// TwinCAT 3 PLC project ArbiterPLC
// ProgramVersion: 3.1.4022.7
// libraries:
//   Tc2_MC2, * (Beckhoff Automation GmbH)
//   Tc2_Standard, * (Beckhoff Automation GmbH)
//   Tc2_System, * (Beckhoff Automation GmbH)
//   Tc2_SystemCX, * (Beckhoff Automation GmbH)
//   Tc2_Utilities, * (Beckhoff Automation GmbH)
//   Tc3_Module, * (Beckhoff Automation GmbH)
//   LCLS General,newest,SLAC
//   PMPS,0.0.0,SLAC - LCLS
// project tree:
//   / FFOTask.TcTTO, PlcTask.TcTTO
//   GVLs/ GVL.TcGVL, GVL_CheckBounds.TcGVL
//   ImplicitChecks/ CheckBounds.TcPOU, CheckRangeSigned.TcPOU, CheckRangeUnsigned.TcPOU
//   POUs/Accelerator/ FB_Hgvpu.TcPOU, FB_SXU.TcPOU, FB_UndulatorSegment.TcPOU
//   POUs/ CurrentBPUpdate.TcPOU, CXDisplay.TcPOU, Fast_Faults_Evaluate.TcPOU, FB_BPControlDevice.TcPOU, FB_eVSimulator.TcPOU, FB_StopperWatcher.TcPOU, MachineSimulation.TcPOU, MAIN.TcPOU, PMPS_Arbiter.TcPOU, Testing.TcPOU
// real-time tasks:
//   TASK PlcTask: cycle T#10ms, priority 2, ADS port 350
//   TASK FFOTask: cycle T#1ms, priority 1, ADS port 351
// I/O:
//   DEVICE Device 1 (EtherCAT), AmsNetId 0.0.0.0.2.1
//     Term 12 (EK1200) [EK1200-5000 EtherCAT Power supply (2A E-Bus)]
//       FFO [EL2202 2Ch. Dig. Output 24V, 0.5A]
//       PMPS_Premp [EL2809 16Ch. Dig. Output 24V, 0.5A]
//       Term 12 (EK1122) [EK1122 2 port EtherCAT junction]
//         Term 13 (EK1100) [EK1100 EtherCAT Coupler (2A E-Bus)]
//           PPS_Stoppers [EL1008 8Ch. Dig. Input 24V, 3ms]
//           Term 15 (EL1008) [EL1008 8Ch. Dig. Input 24V, 3ms]
//           MPS_Relay [EL2004 4Ch. Dig. Output 24V, 0.5A]
//           Term 17 (EL2004) [EL2004 4Ch. Dig. Output 24V, 0.5A]
//           Term 30 (EL9011) [EL9011 End Terminal]
//       Term 22 (EK1110) [EK1110 EtherCAT extension]
//     Box 23 (CU1128) [CU1128 6x EtherCAT junction]
//       plc-lfe-optics [EL6695 EtherCAT Bridge terminal (Secondary)]
//       plc-lfe-motion [EL6695 EtherCAT Bridge terminal (Secondary)]
//       Box 26 (EL6692) [EL6692 EtherCAT Bridge terminal (Secondary)]
//       Box 27 (EL6692) [EL6692 EtherCAT Bridge terminal (Secondary)]
//       Term 28 (CU1128-B) [CU1128 6x EtherCAT junction - Dev A]
//       Term 29 (CU1128-C) [CU1128 6x EtherCAT junction - Dev B]
//       Term 31 (EL9010) [EL9010 End Terminal]
// variable links:
//   ArbiterPLC Instance <-> Device 1 (EtherCAT)
//     PlcTask Inputs/MAIN.fbEcatDiag.arrEcMasterNetId <-> InfoData/AmsNetId
//     PlcTask Inputs/MAIN.fbEcatDiag.nEcMasterDevState <-> Inputs/DevState
//     PlcTask Inputs/MAIN.fbEcatDiag.nEcMasterDeviceId <-> InfoData/DevId
//     PlcTask Inputs/MAIN.fbEcatDiag.nEcMasterSlaveCount <-> Inputs/SlaveCount
//     PlcTask Inputs/MAIN.fbEcatDiag.nEcMasterSlaveCountCfg <-> InfoData/CfgSlaveCount
//   ArbiterPLC Instance <-> Device 1 (EtherCAT)/Box 23 (CU1128)/plc-lfe-motion
//     PlcTask Inputs/PMPS_Arbiter.lfe_PMPS_IO.i_Connected <-> SYNC Inputs/External device not connected
//     PlcTask Inputs/PMPS_Arbiter.lfe_PMPS_IO.i_RequestedBP <-> IO Inputs/RequestedBP
//     PlcTask Inputs/PMPS_Arbiter.lfe_PMPS_IO.i_TxPDOState <-> SYNC Inputs/TxPDO state
//     PlcTask Outputs/PMPS_Arbiter.lfe_PMPS_IO.o_CurrentBP <-> IO Outputs/CurrentBP
//   ArbiterPLC Instance <-> Device 1 (EtherCAT)/Term 12 (EK1200)/PMPS_Premp
//     PlcTask Outputs/PMPS_Arbiter.fbCuInterface.q_CLTS_ASSERTION_LINES[1] <-> Channel 9/Output
//     PlcTask Outputs/PMPS_Arbiter.fbCuInterface.q_CLTS_ASSERTION_LINES[2] <-> Channel 10/Output
//     PlcTask Outputs/PMPS_Arbiter.fbCuInterface.q_CLTS_ASSERTION_LINES[3] <-> Channel 11/Output
//     PlcTask Outputs/PMPS_Arbiter.fbMPSInterface.q_BC_ASSERTION_LINES[{1..8}] <-> Channel {1..8}/Output  (8 links)
//   ArbiterPLC Instance <-> Device 1 (EtherCAT)/Term 12 (EK1200)/Term 12 (EK1122)/Term 13 (EK1100)/MPS_Relay
//     PlcTask Outputs/PMPS_Arbiter.st1l0Watcher.q_StopperIN_Relay <-> Channel 2/ST1L0_RELAY_IN
//     PlcTask Outputs/PMPS_Arbiter.st1l0Watcher.q_StopperOUT_Relay <-> Channel 1/ST1L0_RELAY_OUT
//   ArbiterPLC Instance <-> Device 1 (EtherCAT)/Term 12 (EK1200)/Term 12 (EK1122)/Term 13 (EK1100)/PPS_Stoppers
//     PlcTask Inputs/PMPS_Arbiter.st1l0Watcher.i_StopperInLS <-> Channel 1/ST1L0_PPS_IN
//     PlcTask Inputs/PMPS_Arbiter.st1l0Watcher.i_StopperOutLS <-> Channel 2/ST1L0_PPS_OUT

CONFIGURATION ArbiterPLC
    RESOURCE PLC ON TwinCAT3
        TASK FFOTask(INTERVAL := T#1ms, PRIORITY := 1);
        TASK PlcTask(INTERVAL := T#10ms, PRIORITY := 2);
        PROGRAM Fast_Faults_Evaluate WITH FFOTask : Fast_Faults_Evaluate;
        PROGRAM MAIN WITH PlcTask : MAIN;
    END_RESOURCE
END_CONFIGURATION

// ---- GVLs/GVL.TcGVL

VAR_GLOBAL
   {attribute 'pytmc' := '
    pv: @(PREFIX)Arbiter:01
    '}
	g_fbArbiter1	:	FB_Arbiter(25);

	ReqBP	:	ST_BeamParams; //Currently the placeholder for the fully arbitrated BP set
	
	//Example implementation of the FFO
    
    {attribute 'pytmc' := '
    pv: @(PREFIX)FFO:01
    '}
	{attribute 'TcLinkTo' := '.q_xFastFaultOut:=TIIB[PMPS_FFO]^Channel 1^Output'}
	g_FastFaultOutput1	:	FB_HardwareFFOutput;
    
	g_rTestingVelocity	:	LREAL := PMPS_GVL.VISIBLE_TEST_VELOCITY;
    
    AttemptReset    :   BOOL; // For testing
END_VAR

// ---- GVLs/GVL_CheckBounds.TcGVL
{attribute 'qualified_only'}
VAR_GLOBAL
    nTooLow : UDINT;
    nTooHigh : UDINT;
    nDivByZero : UDINT;
END_VAR

// ---- POUs/Fast_Faults_Evaluate.TcPOU
PROGRAM Fast_Faults_Evaluate
VAR
END_VAR

g_FastFaultOutput1.EvaluateOutput(i_xVeto:=PMPS_GVL.stCurrentBeamParameters.aStoppers[PMPS.L_Stopper.ST1L0]);

END_PROGRAM

// ---- POUs/MAIN.TcPOU
PROGRAM MAIN
VAR
	Initialize	:	BOOL := TRUE;
    
	fbLogHandler : FB_LogHandler;
	fbEcatDiag : FB_EcatDiagWrapper;

	{attribute 'pytmc' := '
		pv: Arbiter:Link:HGVPU
		link: USEG:UNDH:
	'}
	fbHgvpu : FB_Hgvpu;
	
	{attribute 'pytmc' := '
		pv: Arbiter:Link:SXU
		link: USEG:UNDS:
	'}
	fbSxu : FB_SXU;
	
	{attribute 'pytmc' := '
    pv: @(PREFIX)BeamParamCntl
    '}
	fbBPControl : FB_BPControlDevice(nID:=10);

END_VAR

//Arbiter PLC

IF Initialize THEN
	Initialize := FALSE;
END_IF

// Ethercat Diagnostics
fbEcatDiag();

///////////////////////////////////////////////////
// This code should be disabled or removed in deployment
// Might have a switch to change to simulation mode
MachineSimulation();
Testing();
///////////////////////////////////////////////////	

fbHgvpu();
fbSxu();

// Dummy device for controling pmps beam parameters
fbBPControl(Arbiter:=g_fbArbiter1);

//Update current BP
CurrentBPUpdate();

// PMPS Functionality	
PMPS_Arbiter();


fbLogHandler();

ACTION Initialize:

END_ACTION

END_PROGRAM

// ---- POUs/Accelerator/FB_Hgvpu.TcPOU
FUNCTION_BLOCK FB_Hgvpu
VAR_INPUT
	
END_VAR

VAR_OUTPUT
END_VAR


VAR
    // From lcls-srv01: grep -e KDes  /u1/lcls/epics/ioc/data/ioc-undh-uc*/iocInfo/IOC.pvlist |sort

    {attribute 'pytmc' := 'pv: 24; link: 2450:'}
    fbSegment_24 : FB_UndulatorSegment;
    
    {attribute 'pytmc' := 'pv: 25; link: 2550:'}
    fbSegment_25 : FB_UndulatorSegment;
    
    {attribute 'pytmc' := 'pv: 26; link: 2650:'}
    fbSegment_26 : FB_UndulatorSegment;
    
    {attribute 'pytmc' := 'pv: 27; link: 2750:'}
    fbSegment_27 : FB_UndulatorSegment;
    
    {attribute 'pytmc' := 'pv: 29; link: 2950:'}
    fbSegment_29 : FB_UndulatorSegment;
    
    {attribute 'pytmc' := 'pv: 30; link: 3050:'}
    fbSegment_30 : FB_UndulatorSegment;
    
    {attribute 'pytmc' := 'pv: 31; link: 3150:'}
    fbSegment_31 : FB_UndulatorSegment;
    
    {attribute 'pytmc' := 'pv: 32; link: 3250:'}
    fbSegment_32 : FB_UndulatorSegment;
    
    {attribute 'pytmc' := 'pv: 33; link: 3350:'}
    fbSegment_33 : FB_UndulatorSegment;
    
    {attribute 'pytmc' := 'pv: 34; link: 3450:'}
    fbSegment_34 : FB_UndulatorSegment;
    
    {attribute 'pytmc' := 'pv: 35; link: 3550:'}
    fbSegment_35 : FB_UndulatorSegment;
    
    {attribute 'pytmc' := 'pv: 36; link: 3650:'}
    fbSegment_36 : FB_UndulatorSegment;
    
    {attribute 'pytmc' := 'pv: 37; link: 3750:'}
    fbSegment_37 : FB_UndulatorSegment;
    
    {attribute 'pytmc' := 'pv: 38; link: 3850:'}
    fbSegment_38 : FB_UndulatorSegment;
    
    {attribute 'pytmc' := 'pv: 39; link: 3950:'}
    fbSegment_39 : FB_UndulatorSegment;
    
    {attribute 'pytmc' := 'pv: 40; link: 4050:'}
    fbSegment_40 : FB_UndulatorSegment;
    
    {attribute 'pytmc' := 'pv: 41; link: 4150:'}
    fbSegment_41 : FB_UndulatorSegment;
    
    {attribute 'pytmc' := 'pv: 42; link: 4250:'}
    fbSegment_42 : FB_UndulatorSegment;
    
    {attribute 'pytmc' := 'pv: 43; link: 4350:'}
    fbSegment_43 : FB_UndulatorSegment;
    
    {attribute 'pytmc' := 'pv: 44; link: 4450:'}
    fbSegment_44 : FB_UndulatorSegment;
    
    {attribute 'pytmc' := 'pv: 45; link: 4550:'}
    fbSegment_45 : FB_UndulatorSegment;
    
    {attribute 'pytmc' := 'pv: 46; link: 4650:'}
    fbSegment_46 : FB_UndulatorSegment;
    
    fbSegment : ARRAY [iLowBound..iHighBound] OF POINTER TO FB_UndulatorSegment;
    fbCurrentSegment : REFERENCE TO FB_UndulatorSegment;

    iIndex : UDINT;

    bInitialized : BOOL := FALSE;

END_VAR

VAR CONSTANT
    iLowBound  : UDINT := 24;
    iHighBound : UDINT := 46;
END_VAR

IF NOT bInitialized THEN

    fbSegment[24] := ADR(fbSegment_24);
    fbSegment[25] := ADR(fbSegment_25);
    fbSegment[26] := ADR(fbSegment_26);
    fbSegment[27] := ADR(fbSegment_27);
    fbSegment[28] := 0;
    fbSegment[29] := ADR(fbSegment_29);
    fbSegment[30] := ADR(fbSegment_30);
    fbSegment[31] := ADR(fbSegment_31);
    fbSegment[32] := ADR(fbSegment_32);
    fbSegment[33] := ADR(fbSegment_33);
    fbSegment[34] := ADR(fbSegment_34);
    fbSegment[35] := ADR(fbSegment_35);
    fbSegment[36] := ADR(fbSegment_36);
    fbSegment[37] := ADR(fbSegment_37);
    fbSegment[38] := ADR(fbSegment_38);
    fbSegment[39] := ADR(fbSegment_39);
    fbSegment[40] := ADR(fbSegment_40);
    fbSegment[41] := ADR(fbSegment_41);
    fbSegment[42] := ADR(fbSegment_42);
    fbSegment[43] := ADR(fbSegment_43);
    fbSegment[44] := ADR(fbSegment_44);
    fbSegment[45] := ADR(fbSegment_45);
    fbSegment[46] := ADR(fbSegment_46);

    bInitialized := TRUE;
END_IF

FOR iIndex := iLowBound TO iHighBound DO
    IF fbSegment[iIndex] <> 0 THEN
		fbCurrentSegment REF= fbSegment[iIndex]^;
		fbCurrentSegment();
    END_IF
END_FOR

END_FUNCTION_BLOCK

// ---- POUs/Accelerator/FB_UndulatorSegment.TcPOU
FUNCTION_BLOCK FB_UndulatorSegment
VAR_INPUT
END_VAR
VAR_OUTPUT
END_VAR
VAR
	{attribute 'pytmc' := '
		pv: KDes
		link: KDes
	'}
	fbKDesired : FB_LREALFromEPICS;

	{attribute 'pytmc' := '
		pv: KAct
		link: KAct
	'}
	fbKActual : FB_LREALFromEPICS;

END_VAR

fbKDesired();
fbKActual();

END_FUNCTION_BLOCK

// ---- POUs/Accelerator/FB_SXU.TcPOU
FUNCTION_BLOCK FB_SXU
VAR_INPUT
	
END_VAR

VAR_OUTPUT
END_VAR



VAR
    // From lcls-srv01: grep -e KDes  /u1/lcls/epics/ioc/data/sioc-unds-uc*/iocInfo/IOC.pvlist |sort


    {attribute 'pytmc' := 'pv: 26; link: 2650:'}
    fbSegment_26 : FB_UndulatorSegment;
    
    {attribute 'pytmc' := 'pv: 27; link: 2750:'}
    fbSegment_27 : FB_UndulatorSegment;
    
    {attribute 'pytmc' := 'pv: 28; link: 2850:'}
    fbSegment_28 : FB_UndulatorSegment;
    
    {attribute 'pytmc' := 'pv: 29; link: 2950:'}
    fbSegment_29 : FB_UndulatorSegment;
    
    {attribute 'pytmc' := 'pv: 30; link: 3050:'}
    fbSegment_30 : FB_UndulatorSegment;
    
    {attribute 'pytmc' := 'pv: 31; link: 3150:'}
    fbSegment_31 : FB_UndulatorSegment;
    
    {attribute 'pytmc' := 'pv: 32; link: 3250:'}
    fbSegment_32 : FB_UndulatorSegment;
    
    {attribute 'pytmc' := 'pv: 33; link: 3350:'}
    fbSegment_33 : FB_UndulatorSegment;
    
    {attribute 'pytmc' := 'pv: 34; link: 3450:'}
    fbSegment_34 : FB_UndulatorSegment;
    
    {attribute 'pytmc' := 'pv: 36; link: 3650:'}
    fbSegment_36 : FB_UndulatorSegment;
    
    {attribute 'pytmc' := 'pv: 37; link: 3750:'}
    fbSegment_37 : FB_UndulatorSegment;
    
    {attribute 'pytmc' := 'pv: 38; link: 3850:'}
    fbSegment_38 : FB_UndulatorSegment;
    
    {attribute 'pytmc' := 'pv: 39; link: 3950:'}
    fbSegment_39 : FB_UndulatorSegment;
    
    {attribute 'pytmc' := 'pv: 40; link: 4050:'}
    fbSegment_40 : FB_UndulatorSegment;
    
    {attribute 'pytmc' := 'pv: 41; link: 4150:'}
    fbSegment_41 : FB_UndulatorSegment;
    
    {attribute 'pytmc' := 'pv: 42; link: 4250:'}
    fbSegment_42 : FB_UndulatorSegment;
    
    {attribute 'pytmc' := 'pv: 43; link: 4350:'}
    fbSegment_43 : FB_UndulatorSegment;
    
    {attribute 'pytmc' := 'pv: 44; link: 4450:'}
    fbSegment_44 : FB_UndulatorSegment;
    
    {attribute 'pytmc' := 'pv: 45; link: 4550:'}
    fbSegment_45 : FB_UndulatorSegment;
    
    {attribute 'pytmc' := 'pv: 46; link: 4650:'}
    fbSegment_46 : FB_UndulatorSegment;
    
    {attribute 'pytmc' := 'pv: 47; link: 4750:'}
    fbSegment_47 : FB_UndulatorSegment;
    


    fbSegment : ARRAY [iLowBound..iHighBound] OF POINTER TO FB_UndulatorSegment;
    fbCurrentSegment : REFERENCE TO FB_UndulatorSegment;

    iIndex : UDINT;

    bInitialized : BOOL := FALSE;

END_VAR

VAR CONSTANT
    iLowBound  : UDINT := 26;
    iHighBound : UDINT := 47;
END_VAR



IF NOT bInitialized THEN

    fbSegment[26] := ADR(fbSegment_26);
    fbSegment[27] := ADR(fbSegment_27);
    fbSegment[28] := ADR(fbSegment_28);
    fbSegment[29] := ADR(fbSegment_29);
    fbSegment[30] := ADR(fbSegment_30);
    fbSegment[31] := ADR(fbSegment_31);
    fbSegment[32] := ADR(fbSegment_32);
    fbSegment[33] := ADR(fbSegment_33);
    fbSegment[34] := ADR(fbSegment_34);
    fbSegment[35] := 0;
    fbSegment[36] := ADR(fbSegment_36);
    fbSegment[37] := ADR(fbSegment_37);
    fbSegment[38] := ADR(fbSegment_38);
    fbSegment[39] := ADR(fbSegment_39);
    fbSegment[40] := ADR(fbSegment_40);
    fbSegment[41] := ADR(fbSegment_41);
    fbSegment[42] := ADR(fbSegment_42);
    fbSegment[43] := ADR(fbSegment_43);
    fbSegment[44] := ADR(fbSegment_44);
    fbSegment[45] := ADR(fbSegment_45);
    fbSegment[46] := ADR(fbSegment_46);
    fbSegment[47] := ADR(fbSegment_47);

    bInitialized := TRUE;
END_IF

FOR iIndex := iLowBound TO iHighBound DO
    IF fbSegment[iIndex] <> 0 THEN
		fbCurrentSegment REF= fbSegment[iIndex]^;
		fbCurrentSegment();
    END_IF
END_FOR

END_FUNCTION_BLOCK

// ---- POUs/FB_BPControlDevice.TcPOU
(*
Used to request a beam parameter set from EPICS.

Technically just one of these is needed in the entire
PMPS for a line.

*)
FUNCTION_BLOCK FB_BPControlDevice
VAR_INPUT
END_VAR
VAR_OUTPUT
END_VAR
VAR_IN_OUT
	Arbiter : FB_Arbiter;
END_VAR
VAR
	{attribute 'pytmc' := '
    	pv: ReqBP
		io: o
    '}
	EpicsReqBP : ST_BeamParams;
	{attribute 'pytmc' := '
    	pv: Apply
		io: o
    '}
	bApply : BOOL;
	
	nControlDeviceID : DWORD;
	
	rtApply : R_TRIG;
	
END_VAR


rtApply(CLK:=bApply);
IF rtApply.Q THEN
	Arbiter.RemoveRequest(nControlDeviceID);
	Arbiter.AddRequest(nControlDeviceID, EpicsReqBP);
	bApply := FALSE;
END_IF

METHOD FB_init : BOOL
VAR_INPUT
	bInitRetains : BOOL; // if TRUE, the retain variables are initialized (warm start / cold start)
	bInCopyCode : BOOL;  // if TRUE, the instance afterwards gets moved into the copy code (online change)
	nID : DWORD := PMPS_GVL.EXCLUDED_ASSERTION_ID;
END_VAR
nControlDeviceID:= nID;
END_METHOD

END_FUNCTION_BLOCK

// ---- POUs/MachineSimulation.TcPOU
PROGRAM MachineSimulation
VAR
	fbMachine	:	FB_MachineSimulator; //Simulates attenuator as well
	fbeVSimulator : FB_eVSimulator := (NoiseLevel := 1);
END_VAR

// reV Simulator
fbeVSimulator();

// Machine simulator
fbMachine(
	i_stAssertedParams := PMPS_GVL.stRequestedBeamParameters,
	q_stMachineParams => PMPS_GVL.stCurrentBeamParameters,
	i_xFault	:= NOT GVL.g_FastFaultOutput1.q_xFastFaultOut
	);

PMPS_GVL.stCurrentBeamParameters.neVRange := F_eVRangeCalculator(fbeVSimulator.eV, PMPS_GVL.stCurrentBeamParameters.neVRange);

END_PROGRAM

// ---- POUs/FB_eVSimulator.TcPOU
(* eV Simulator
A. Wallace 2019-8-30

Adds noise to the eV and changes eV position occasionally.
*)
FUNCTION_BLOCK FB_eVSimulator
VAR_INPUT
	NoiseLevel	:	REAL	:= 0; // eV Noise
	ChangeTime : TIME := T#10S;
END_VAR
VAR_OUTPUT
	eV	:	REAL := 300;
END_VAR
VAR
	eVRange : REAL := 1600;
	timer: TON;
	eVRand	:	DRAND :=(Seed:=0);
	NoiseRand : DRAND := (Seed:=0);
END_VAR


timer(in:=TRUE, PT:=ChangeTime);

//Occasionally change eV
IF timer.Q THEN
	timer(in:=FALSE);
	eVRand();
	eV := LIMIT(0, eVRange*LREAL_TO_REAL(eVRand.Num), eVRange);
END_IF

// Noise generation
NoiseRand();
eV := eV + NoiseLevel*LREAL_TO_REAL(NoiseRand.Num);
NoiseRand();
eV := LIMIT(0, ev - NoiseLevel*LREAL_TO_REAL(NoiseRand.Num), eVRange);

END_FUNCTION_BLOCK

// ---- POUs/Testing.TcPOU
PROGRAM Testing
VAR
    AttemptReset : TON := (PT:=T#1s);
    gAttemptReset : TON := (PT:=T#500ms);
        
    testFF : FB_FastFault;
    cycle : INT;
END_VAR


// Trip a fast fault periodically
testFF(io_fbFFHWO:= g_FastFaultOutput1);
//testFF.i_xOK := (cycle mod 1000) = 0;
//cycle := cycle + 1;

//Periodically try to reset the photon energy fault.
AttemptReset(IN:=PMPS_Arbiter.fbPhotonEnergyWatcher.xPhotonEnergyWithinBounds, Q=>GVL.AttemptReset);

gAttemptReset(IN:=GVL.g_FastFaultOutput1.xOK, Q=>GVL.g_FastFaultOutput1.i_xReset);

END_PROGRAM

// ---- POUs/PMPS_Arbiter.TcPOU
PROGRAM PMPS_Arbiter
VAR
    
	fbBPRequestor : FB_BPRequestor; // Updates global PMPS RequestedBeamParams
    
	fbPhotonEnergyWatcher	:	FB_PhotonEnergyWatcher;
	{attribute 'pytmc' := '
    pv: @(PREFIX)BeamClassOutputs
    '}
	fbMPSInterface	:	FB_BeamClassOutputs;
    {attribute 'pytmc' := '
    pv: @(PREFIX)CuRateOutputs
    '}
    fbCuInterface	:	FB_CTLS_Outputs;
	
	// Stoppers
	
	{attribute 'TcLinkTo' := '
				.i_StopperInLS:=TIIB[PPS_Stoppers]^Channel 1^ST1L0_PPS_IN;
				.i_StopperOutLS:=TIIB[PPS_Stoppers]^Channel 2^ST1L0_PPS_OUT;
				.q_StopperOUT_Relay:=TIIB[MPS_Relay]^Channel 1^ST1L0_RELAY_OUT;
				.q_StopperIN_Relay:=TIIB[MPS_Relay]^Channel 2^ST1L0_RELAY_IN; 
                                '}
	st1l0Watcher : FB_StopperWatcher(
		PMPS.L_Stopper.ST1L0,
		'ST1L0');
	
	(* Subsystem requests use this FB and a pragma link to pass their requests to the arbiter.
	The fb is called on each cycle and updates the arbiter with the current BP set requested 
	from the subsystem PLC.*)
	//<TODO> make this so it does input and output to the IF
    (*{attribute 'pytmc' := '
    pv: @(PREFIX):PLC1
    '}*)
	{attribute 'TcLinkTo' := '.i_RequestedBP:=TIIB[plc-lfe-motion]^IO Inputs^RequestedBP; 
                                .o_CurrentBP:=TIIB[plc-lfe-motion]^IO Outputs^CurrentBP;
                                .i_Connected:=TIIB[plc-lfe-motion]^SYNC Inputs^External device not connected;
                                .i_WcState:=TIIB[plc-lfe-motion]^WcState^WcState;
                                .i_TxPDOState:=TIIB[plc-lfe-motion]^SYNC Inputs^TxPDO state;
                                '}
	lfe_PMPS_IO : FB_ArbiterToSubSys_IO := (RequestingSystemID := 16#FF0F);
    
	(*{attribute 'pytmc' := '
    pv: @(PREFIX)SubSysIO:PLC2
    '}*)
	{attribute 'TcLinkTo' := '.i_RequestedBP:=TIIB[SubSysPLC2]^IO Inputs^RequestedBP;
                                .i_xNewRequest:=TIIB[SubSysPLC2]^IO Inputs^xNewRequest; 
                                .o_CurrentBP:=TIIB[SubSysPLC2]^IO Outputs^CurrentBP;
                                .i_Connected:=TIIB[SubSysPLC2]^SYNC Inputs^External device not connected;
                                .i_WcState:=TIIB[SubSysPLC2]^WcState^WcState;
                                .i_TxPDOState:=TIIB[SubSysPLC2]^SYNC Inputs^TxPDO state;
                                .i_TxPDOToggle:=TIIB[SubSysPLC2]^SYNC Inputs^TxPDO toggle;
                                '}
	//fbSubSys2_PMPS_IO : FB_ArbiterToSubSys_IO := (RequestingSystemID := 16#FF10);
    
    
	
END_VAR


// Watching stopper statuses
st1l0Watcher();

// Updating arbiter with subsystem requests.
lfe_PMPS_IO(Arbiter:=GVL.g_fbArbiter1, fbFFHWO:=GVL.g_FastFaultOutput1, Reset:=GVL.AttemptReset);

//fbSubSys2_PMPS_IO(Arbiter:=GVL.g_fbArbiter1, fbFFHWO:=GVL.g_FastFaultOutput1, Reset:=GVL.AttemptReset);

// Example with attenuator peel-off
//////////////////////////////////

// Beam parameter requestor
fbBPRequestor(Arbiter:=GVL.g_fbArbiter1, q_ReqBP => PMPS_GVL.stRequestedBeamParameters);

// Request beam class
fbMPSInterface(BP := PMPS_GVL.stRequestedBeamParameters);

// Request Cu beam rate
fbCuInterface(BP := PMPS_GVL.stRequestedBeamParameters);


// Keep an eye on the photon energy
fbPhotonEnergyWatcher(i_stCurrentBeamParams	:= PMPS_GVL.stCurrentBeamParameters,
					i_stRequestedBeamParams := PMPS_GVL.stRequestedBeamParameters,
					io_fbFFHWO:= GVL.g_FastFaultOutput1,
                    i_xReset := GVL.AttemptReset);

// Evaluate fast fault vetos
g_FastFaultOutput1.EvaluateOverrides();

// Send fast fault logs
g_FastFaultOutput1.ExecuteLogging();

END_PROGRAM

// ---- POUs/FB_StopperWatcher.TcPOU
// Relays stopper state and sends a message when stopper state changes.
FUNCTION_BLOCK FB_StopperWatcher
VAR_INPUT
END_VAR
VAR_OUTPUT
END_VAR
VAR
	i_StopperOutLS AT %I* : BOOL;
	i_StopperInLS AT %I* : BOOL;
	
	q_StopperOUT_Relay AT %Q* : BOOL;
	q_StopperIN_Relay AT %Q* : BOOL;
	
	eStopper : PMPS.L_Stopper;
	StopperName : STRING;
	
	// Logging
	fbLogMsg : FB_LogMessage := (
		eSubSystem := E_Subsystem.MPS);
		
	rtIn : R_TRIG;
	rtOut : R_TRIG;
	
END_VAR


rtIn(CLK := i_StopperInLS);
rtOut(CLK := i_StopperOutLS);

IF rtIn.Q THEN
	fbLogMsg.sMsg := CONCAT(StopperName, ' moved IN');
	fbLogMsg();
ELSIF rtOut.Q THEN
	fbLogMsg.sMsg := CONCAT(StopperName, ' moved OUT');
	fbLogMsg();
END_IF

q_StopperOUT_Relay := i_StopperOutLS;
q_StopperIN_Relay := i_StopperInLS;

METHOD FB_init : BOOL
VAR_INPUT
	bInitRetains : BOOL; // if TRUE, the retain variables are initialized (warm start / cold start)
	bInCopyCode : BOOL;  // if TRUE, the instance afterwards gets moved into the copy code (online change)
	Stopper : PMPS.L_Stopper;
	sStopperName : STRING;
END_VAR
eStopper := Stopper;
StopperName := sStopperName;
END_METHOD

END_FUNCTION_BLOCK

// ---- POUs/CurrentBPUpdate.TcPOU
PROGRAM CurrentBPUpdate
VAR
END_VAR

END_PROGRAM

// ---- ImplicitChecks/CheckBounds.TcPOU
// Implicitly generated code : DO NOT EDIT
FUNCTION CheckBounds : DINT
VAR_INPUT
	index, lower, upper: DINT;
END_VAR
// User defined local variables
VAR
    sMessageLow   : STRING := 'CheckBounds: Index too low (%d)';
    sMessageHigh  : STRING := 'CheckBounds: Index too high (%d)';
END_VAR

// Index too low
IF index < lower THEN
    CheckBounds := lower;
    // Increase global counter
    GVL_CheckBounds.nTooLow := GVL_CheckBounds.nTooLow + 1;
    // Log message
    ADSLOGDINT(msgCtrlMask := ADSLOG_MSGTYPE_WARN,
               msgFmtStr   := sMessageLow,
               dintArg     := index);

// Index too high
ELSIF index > upper THEN
    CheckBounds := upper;
    // Increase global counter
    GVL_CheckBounds.nTooHigh := GVL_CheckBounds.nTooHigh + 1;
    // Log message
    ADSLOGDINT(msgCtrlMask := ADSLOG_MSGTYPE_WARN,
               msgFmtStr   := sMessageHigh,
               dintArg     := index);

// Index OK
ELSE 
    CheckBounds := index;
END_IF
{flow}

END_FUNCTION

// ---- ImplicitChecks/CheckRangeSigned.TcPOU
// Implicitly generated code : DO NOT EDIT
FUNCTION CheckRangeSigned : DINT
VAR_INPUT
	value, lower, upper: DINT;
END_VAR

// Implicitly generated code : Only an Implementation suggestion

IF (value < lower) THEN
	CheckRangeSigned := lower;
ELSIF(value > upper) THEN
	CheckRangeSigned := upper;
ELSE
	CheckRangeSigned := value;
END_IF
{flow}

END_FUNCTION

// ---- ImplicitChecks/CheckRangeUnsigned.TcPOU
// Implicitly generated code : DO NOT EDIT
FUNCTION CheckRangeUnsigned : UDINT
VAR_INPUT
	value, lower, upper: UDINT;
END_VAR

// Implicitly generated code : Only an Implementation suggestion
{noflow}
IF (value < lower) THEN
	CheckRangeUnsigned := lower;
ELSIF(value > upper) THEN
	CheckRangeUnsigned := upper;
ELSE
	CheckRangeUnsigned := value;
END_IF
{flow}

END_FUNCTION

// ---- POUs/CXDisplay.TcPOU
PROGRAM CXDisplay
VAR
    DisplayStats : FB_CXSetTextDisplayUSB := (nPort:=28928);
    fbFormat   : FB_FormatString;
    bError     : BOOL;
    nErrID     : UDINT;
    sOut       : T_MaxString;   
END_VAR

(*
DisplayStats.bExecute S= NOT DisplayStats.bBusy AND NOT DisplayStats.bError;
DisplayStats.bExecute R= DisplayStats.bBusy OR DisplayStats.bError;

DisplayStats.sLine1 := 'PMPS-ARBITER-K';
fbFormat(sFormat := 'Fast Faults: %d', arg1:=F_ULINT(PMPS_GVL.AccumulatedFF), sOut=>DisplayStats.sLine2, bError => bError, nErrID => nErrID ); 

DisplayStats(eMode:=E_CX2100_DisplayModesWr.eCX2100_WriteLines);
*)

END_PROGRAM
